{attribute 'GeneratedUsingTerminal: EL3773-0000-0018'}
{attribute addProperty BoxType "EL3773-0000-0018"}
{attribute addProperty Id "Sample_CountAT %I*UINT2"}
{attribute addProperty CRC "3934833369"}
{attribute addProperty Size "2"}
TYPE AI_Sample_Count_EA88CAD9 :
STRUCT
	{attribute addProperty Name "Sample_Count"}
	Sample_Count AT %I* : UINT;
END_STRUCT
END_TYPE

(* stored: Version 1.2.0.0, ProductVersion 3.1.4024.9
   DUT AI_Sample_Count_EA88CAD9: Id {bce168c1-e491-4b3a-bdd7-8573177e8f24} *)
